Fanuc KAREL source: kt00216.KL

PROGRAM KT00216
%STACKSIZE=65535
%PRIORITY=65535
%NOLOCKGROUP
VAR
OUT : INTEGER
-- UNRESOLVED DECLARATIONS (source type spelling not recovered)
-- Y1 : ARRAY[2] OF TYPE_0x0018 (type_u16=0x2018)
-- H2 : ARRAY[2] OF TYPE_0x0017 (type_u16=0x2017)
BEGIN
Y1[1]=2
-- UNRESOLVED_PC line 9 opcodes [2E 22 9D 33 B4] marker_code=19
-- UNRESOLVED_PC line 10 opcodes [22 9D 33 B1 22 9D 33 B3 46 23] marker_code=38
END KT00216
